// TIA Portal V17 export
ScreenPopup "Codex_Popup_500x500"  500x500
  ScreenLayer 
    TextField "Codex_Popup_Title" at 50,40 size 400x40  Text="Popup 500x500"
